// TIA Portal V19 export
DATA_BLOCK "AUTO ALARM DB"   // DB70
{ S7_Optimized_Access := 'TRUE' }
// stored: MemoryReserve 100
   VAR
      "MFG PROCESS" : Struct
         "PURIFIED WATER PROCESS SELECT" : Bool;
         "PURIFIED WATER PROCESS OF INITIAL DRAIN SELECT" : Bool;
         "PURIFIED WATER PROCESS OF LOAD CELL" : Bool;
         "PURIFIED WATER HEATING OR COOLING SELECT" : Bool;
         "PURIFIED WATER PROCESS OF JACKET DRAIN SELECT" : Bool;
         "PURIFIED WATER PROCESS OVER" : Bool;
         "MATERIAL ADDITION PROCESS SELECT" : Bool;
         "MATERIAL ADDITION MATERIAL ADDED TEXT" : Bool;
         "MATERIAL ADDITION DO YOU WANT TO ADD SORBITOL SELECT" : Bool;
         "MATERIAL ADDITION OF SORBITOL OVER" : Bool;
         "MATERIAL ADDITION DO YOU WANT TO ADD GLUCOSE SELECT" : Bool;
         "MATERIAL ADDITION OF GLUCOSE OVER" : Bool;
         "MATERIAL ADDITION PROCESS OVER" : Bool;
         "RECIRCULATION PROCESS SELECT" : Bool;
         "RECIRCULATION PROCESS RUNING" : Bool;
         "RECIRCULATION OVER" : Bool;
         "MFG PROCESS OVER" : Bool;
      END_STRUCT;
      "MFG PROCESS ALARM" : Struct
         "MFG PROCESS START" : Bool;
         "PURIFIED WATER PROCESS START" : Bool;
         "PURIFIED WATER PROCESS OF INITIAL DRAIN START" : Bool;
         "PURIFIED WATER PROCESS OF INITIAL DRAIN STOP" : Bool;
         "PURIFIED WATER PROCESS OF LOAD CELL START" : Bool;
         "PURIFIED WATER PROCESS OF LOAD CELL STOP" : Bool;
         "PURIFIED WATER OF HEATING START" : Bool;
         "PURIFIED WATER OF HEATING STOP" : Bool;
         "PURIFIED WATER OF COOLING START" : Bool;
         "PURIFIED WATER OF COOLING STOP" : Bool;
         "PURIFIED WATER PROCESS OF JACKET DRAIN START" : Bool;
         "PURIFIED WATER PROCESS OF JACKET DRAIN STOP" : Bool;
         "PURIFIED WATER PROCESS OVER" : Bool;
         "MATERIAL ADDITION PROCESS START" : Bool;
         "MATERIAL ADDITION MATERIAL ADDED TEXT" : Bool;
         "MATERIAL ADDITION OF SORBITOL START" : Bool;
         "MATERIAL ADDITION OF SORBITOL OVER" : Bool;
         "MATERIAL ADDITION OF GLUCOSE START" : Bool;
         "MATERIAL ADDITION OF GLUCOSE OVER" : Bool;
         "MATERIAL ADDITION PROCESS OVER" : Bool;
         "RECIRCULATION PROCESS START" : Bool;
         "RECIRCULATION PROCESS OVER" : Bool;
         "MFG PROCESS OVER" : Bool;
      END_STRUCT;
      "MFG TRANSFER START" : Struct
         "MFG TO STORAGE-1 WITH INLINE HOMO" : Bool;
         "MFG TO STORAGE-1 WITH INLINE FILTER PRES" : Bool;
         "MFG TO STORAGE-2 WITH INLINE HOMO" : Bool;
         "MFG TO STORAGE-2 WITH INLINE FILTER PRES" : Bool;
         "MFG TO STORAGE-3 WITH INLINE HOMO" : Bool;
         "MFG TO STORAGE-3 WITH INLINE FILTER PRES" : Bool;
      END_STRUCT;
      "MFG TRANSFER OVER" : Struct
         "TRANSFER START_MFG TO STORAGE ALL IN ONE FOR OVER (POPUP)" : Bool;
         "MFG TO STORAGE-1 WITH INLINE HOMO" : Bool;
         "MFG TO STORAGE-1 WITH INLINE FILTER PRES" : Bool;
         "MFG TO STORAGE-2 WITH INLINE HOMO" : Bool;
         "MFG TO STORAGE-2 WITH INLINE FILTER PRES" : Bool;
         "MFG TO STORAGE-3 WITH INLINE HOMO" : Bool;
         "MFG TO STORAGE-3 WITH INLINE FILTER PRES" : Bool;
      END_STRUCT;
      "MFG MATERIAL SUCTION" : Struct
         "MATERIAL SUCTION START" : Bool;
         "MATERIAL SUCTION OVER" : Bool;
      END_STRUCT;
      "PREMIXING PROCESS" : Struct
         "PURIFIED WATER PROCESS SELECT" : Bool;
         "PURIFIED WATER PROCESS OF INITIAL DRAIN SELECT" : Bool;
         "PURIFIED WATER PROCESS OF LOAD CELL" : Bool;
         "PURIFIED WATER HEATING OR COOLING SELECT" : Bool;
         "PURIFIED WATER PROCESS OF JACKET DRAIN SELECT" : Bool;
         "PURIFIED WATER PROCESS OVER" : Bool;
         "MATERIAL ADDITION PROCESS SELECT" : Bool;
         "MATERIAL ADDITION MATERIAL ADDED TEXT" : Bool;
         "MATERIAL ADDITION DO YOU WANT TO ADD SORBITOL SELECT" : Bool;
         "MATERIAL ADDITION OF SORBITOL OVER" : Bool;
         "MATERIAL ADDITION DO YOU WANT TO ADD GLUCOSE SELECT" : Bool;
         "MATERIAL ADDITION OF GLUCOSE OVER" : Bool;
         "MATERIAL ADDITION PROCESS OVER" : Bool;
         "RECIRCULATION PROCESS SELECT" : Bool;
         "RECIRCULATION PROCESS RUNING" : Bool;
         "RECIRCULATION OVER" : Bool;
         "PREMIXING PROCESS OVER" : Bool;
      END_STRUCT;
      "PREMIXING PROCESS ALARM" : Struct
         "PREMIXING PROCESS START" : Bool;
         "PURIFIED WATER PROCESS START" : Bool;
         "PURIFIED WATER PROCESS OF INITIAL DRAIN START" : Bool;
         "PURIFIED WATER PROCESS OF INITIAL DRAIN STOP" : Bool;
         "PURIFIED WATER PROCESS OF LOAD CELL START" : Bool;
         "PURIFIED WATER PROCESS OF LOAD CELL STOP" : Bool;
         "PURIFIED WATER OF HEATING START" : Bool;
         "PURIFIED WATER OF HEATING STOP" : Bool;
         "PURIFIED WATER OF COOLING START" : Bool;
         "PURIFIED WATER OF COOLING STOP" : Bool;
         "PURIFIED WATER PROCESS OF JACKET DRAIN START" : Bool;
         "PURIFIED WATER PROCESS OF JACKET DRAIN STOP" : Bool;
         "PURIFIED WATER PROCESS OVER" : Bool;
         "MATERIAL ADDITION PROCESS START" : Bool;
         "MATERIAL ADDITION OF INITIAL DRAIN START" : Bool;
         "MATERIAL ADDITION OF INITIAL DRAIN STOP" : Bool;
         "MATERIAL ADDITION MATERIAL ADDED TEXT" : Bool;
         "MATERIAL ADDITION OF SORBITOL START" : Bool;
         "MATERIAL ADDITION OF SORBITOL OVER" : Bool;
         "MATERIAL ADDITION OF GLUCOSE START" : Bool;
         "MATERIAL ADDITION OF GLUCOSE OVER" : Bool;
         "MATERIAL ADDITION PROCESS OF JACKET DRAIN SELECT" : Bool;
         "MATERIAL ADDITION PROCESS OF JACKET DRAIN STOP" : Bool;
         "MATERIAL ADDITION PROCESS OVER" : Bool;
         "RECIRCULATION PROCESS START" : Bool;
         "RECIRCULATION PROCESS OF INITIAL DRAIN START" : Bool;
         "RECIRCULATION PROCESS OF INITIAL DRAIN STOP" : Bool;
         "RECIRCULATION START" : Bool;
         "RECIRCULATION STOP" : Bool;
         "RECIRCULATION PROCESS OF JACKET DRAIN SELECT" : Bool;
         "RECIRCULATION PROCESS OF JACKET DRAIN STOP" : Bool;
         "RECIRCULATION PROCESS OVER" : Bool;
         "PREMIXING PROCESS OVER" : Bool;
      END_STRUCT;
      "PREMIXING TRANSFER START" : Struct
         "PREMIXING TO MFG WITH INLINE HOMO" : Bool;
         "PREMIXING TO MFG WITH INLINE FILTER PRES" : Bool;
         "PREMIXING TO STORAGE-4 WITH INLINE HOMO" : Bool;
         "PREMIXING TO STORAGE-4 WITH INLINE FILTER PRES" : Bool;
      END_STRUCT;
      "PREMIXING TRANSFER OVER" : Struct
         "PREMIXING TO MFG & STORAGE ALL IN ONE FOR OVER (POPUP)" : Bool;
         "PREMIXING TO MFG WITH INLINE HOMO" : Bool;
         "PREMIXING TO MFG WITH INLINE FILTER PRES" : Bool;
         "PREMIXING TO STORAGE-4 WITH INLINE HOMO" : Bool;
         "PREMIXING TO STORAGE-4 WITH INLINE FILTER PRES" : Bool;
      END_STRUCT;
      "PREMIXING MATERIAL SUCTION" : Struct
         "MATERIAL SUCTION START" : Bool;
         "MATERIAL SUCTION OVER" : Bool;
      END_STRUCT;
      "SUGAR PROCESS" : Struct
         "PURIFIED WATER PROCESS SELECT" : Bool;
         "PURIFIED WATER PROCESS OF INITIAL DRAIN SELECT" : Bool;
         "PURIFIED WATER PROCESS OF LOAD CELL" : Bool;
         "PURIFIED WATER HEATING OR COOLING SELECT" : Bool;
         "PURIFIED WATER PROCESS OF JACKET DRAIN SELECT" : Bool;
         "PURIFIED WATER PROCESS OVER" : Bool;
         "MFG PROCESS OVER" : Bool;
      END_STRUCT;
      "SUGAR PROCESS ALARM" : Struct
         "SUGAR PROCESS START" : Bool;
         "PURIFIED WATER PROCESS START" : Bool;
         "PURIFIED WATER PROCESS OF INITIAL DRAIN START" : Bool;
         "PURIFIED WATER PROCESS OF INITIAL DRAIN STOP" : Bool;
         "PURIFIED WATER PROCESS OF LOAD CELL START" : Bool;
         "PURIFIED WATER PROCESS OF LOAD CELL STOP" : Bool;
         "PURIFIED WATER OF HEATING START" : Bool;
         "PURIFIED WATER OF HEATING STOP" : Bool;
         "PURIFIED WATER OF COOLING START" : Bool;
         "PURIFIED WATER OF COOLING STOP" : Bool;
         "PURIFIED WATER PROCESS OF JACKET DRAIN START" : Bool;
         "PURIFIED WATER PROCESS OF JACKET DRAIN STOP" : Bool;
         "PURIFIED WATER PROCESS OVER" : Bool;
      END_STRUCT;
      "SUGAR TRANSFER START" : Struct
         "SUGAR TRANSFER SELECT POPUP" : Bool;
         "TRANSFER PREMIXING AND MFG POPUP" : Bool;
         "SUGAR TO PREMIXING" : Bool;
         "SUGAR TO MFG" : Bool;
      END_STRUCT;
      "SUGAR TRANSFER OVER" : Struct
         "SUGAR TRANSFER OVER POPUP" : Bool;
         "SUGAR TO PREMIXING" : Bool;
         "SUGAR TO MFG" : Bool;
      END_STRUCT;
      "SUGAR MATERIAL SUCTION" : Struct
         "MATERIAL SUCTION START" : Bool;
         "MATERIAL SUCTION OVER" : Bool;
      END_STRUCT;
   END_VAR
BEGIN
END_DATA_BLOCK
